{attribute 'GeneratedUsingTerminal: EL1502--0000'}
{attribute addProperty BoxType "EL1502--0000"}
{attribute addProperty Id "CNT_InputsAT %I*CNT_Inputs_7D4495CD11CNT_OutputsAT %Q*CNT_Outputs_EB14A6758WcStateAT %I*WcState_9091E0EB2InfoDataAT %I*InfoData_94A18F5E2"}
{attribute addProperty CRC "2212941383"}
{attribute addProperty Size "23"}
TYPE EL1502_83E6CE47 EXTENDS EtcSlaveTerminalBase_947E5A46 :
STRUCT
	{attribute addProperty Name "CNT_Inputs"}
	CNT_Inputs : CNT_Inputs_7D4495CD;
	{attribute addProperty Name "CNT_Outputs"}
	CNT_Outputs : CNT_Outputs_EB14A675;
	{attribute addProperty Name "WcState"}
	WcState : WcState_9091E0EB;
	{attribute addProperty Name "InfoData"}
	InfoData : InfoData_94A18F5E;
END_STRUCT
END_TYPE

(* stored: Version 1.2.0.0, ProductVersion 3.1.4024.9
   DUT EL1502_83E6CE47: Id {8dca4d24-3ae7-48e9-ba09-858841540753} *)
